(* CODESYS project øving 3.ecp

Project tree, tasks and I/O mapping:
  Controller : 750-8214 PFC200 G2 2ETH RS CAN, WAGO, order no. 0750-8214, version 5.16.3.16
    application Application
      libraries: 
      task PLC_Task (cyclic, interval t#50ms, priority 15) calls PLC_PRG, Oppgave4Teller, Oppgave3ST, Oppgave2BTest, Oppgave2ST
      task VISU_TASK (cyclic, interval 100 ms, priority 15) calls VisuElems.Visu_Prg
      program PLC_PRG [ST]
      global variables GVL
      Oppgave2/
        program Oppgave2ALD [LD]
        program Oppgave2ST [ST]
        program Oppgave2FBD [FBD]
        function Oppgave2A [FBD]
        function MFTest [FBD]
        function MLTest [LD]
        function MSTest [ST]
        function block RTF [FBD]
      Oppgave3/
        program Oppgave3LD [FBD]
        program Oppgave3FBD [FBD]
        program Oppgave3ST [FBD]
        function block Oppgave3STD [ST]
        function block Oppgave3FBDD [FBD]
        function block Oppgave3LDD [LD]
        visualisation Oppgave3GUI
      Oppgave4/
        function block Oppgave4Timeteller [ST]
        program Oppgave4Teller [FBD]
        visualisation Oppgave4Meny
      Oppgave2B/
        function Oppgave2B [ST]
        program Oppgave2BTest [ST]
      Oppgave1/
        program Oppgave1 [ST]
    ProjectConfigurationTxt
    ProjectConfiguration
    Kbus : Kbus, WAGO, version 1.4.0.2
        unmapped channels: K-BUS diagnostics
    MODBUS
      MODBUS : MODBUS, WAGO, order no. n/a, version 1.1.1.16
    CANbus
    Common.PCI
    EtherNet/IP
      Ethernet : Ethernet, WAGO, version 35.16.0.0
    Serial
      COM1 : COM1, WAGO, version 0.0.0.19
  00000000-0000-0000-0000-000000000000|C:\Users\kjebo\AppData\Local\Temp\4e63b915f46a404b8f25f3cc1ab48cd9\ProjectCfg.txt
  00000000-0000-0000-0000-000000000000|C:\Users\kjebo\AppData\Local\Temp\8f733436873c440eb71a6538c97844ea\Project.xml
  text list GlobalTextList
*)

// Controller/Application/GVL
{attribute 'qualified_only'}
VAR_GLOBAL
	Majority: BOOL;
	Vote1: BOOL;
	Vote2: BOOL;
	Vote3: BOOL;
	Trig: BOOL;
	Inn: BOOL;
	Ut: BOOL;
	
END_VAR

// Controller/Application/PLC_PRG
PROGRAM PLC_PRG
VAR
END_VAR

END_PROGRAM

// Controller/Application/Oppgave4/Oppgave4Teller
PROGRAM Oppgave4Teller
VAR
	Kjorer : BOOL;
	Time_ell: TIME;
	Timeteller_1: Oppgave4Timeteller;
	Omstart: BOOL;
	Alarm: BOOL; 
END_VAR

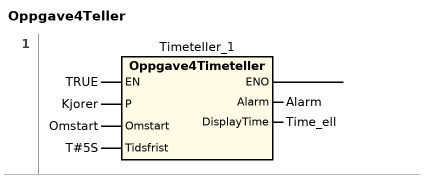
// NETWORK 1
Timeteller_1(P := Kjorer, Omstart := Omstart, Tidsfrist := T#5S, Alarm => Alarm, DisplayTime => Time_ell); // Oppgave4Timeteller

END_PROGRAM

// Controller/Application/Oppgave4/Oppgave4Timeteller
FUNCTION_BLOCK Oppgave4Timeteller
VAR_INPUT
	P: BOOL;
	Omstart: BOOL;
	Tidsfrist: TIME;
END_VAR
VAR_OUTPUT
	Alarm: BOOL;
	DisplayTime : TIME;
END_VAR
VAR
	T: TIME;
	T0: TIME;
	TT: TIME;
	StartTime: TIME;
	On: BOOL;
	P_A: BOOL;
	P_0: BOOL;
	Stopp: TIME;
	TotalRun : TIME;
	Sekunder: TIME;
END_VAR

P_A := P AND NOT (P_0);
P_0 := P;


//IF T0 = TIME() - TIME() THEN
	//T0 := TIME();
//END_IF
T := TIME();
IF On THEN
	//TT := TT + (T-T0);
	Sekunder := T - StartTime;
	IF T > Stopp THEN
		On := FALSE;
		TotalRun := Sekunder + TotalRun;
		Sekunder := T#0S;
		
	END_IF
ELSE 
	IF P_A THEN
		StartTime := T;
		TotalRun := Sekunder + TotalRun;
		Sekunder := T#0S;
		Stopp := StartTime + Tidsfrist;
		On := TRUE;
	END_IF
	
END_IF
T0 := T;
Displaytime := TotalRun + Sekunder;

IF T >= Stopp THEN
	Alarm := TRUE;
ELSE
	Alarm := FALSE;
END_IF

// Reset
IF Omstart THEN
	DisplayTime := T#0S;
	TotalRun := T#0s;
END_IF

END_FUNCTION_BLOCK

// Controller/Application/Oppgave3/Oppgave3ST
PROGRAM Oppgave3ST
VAR
	Oppgave3ST_0: Oppgave3STD;
END_VAR

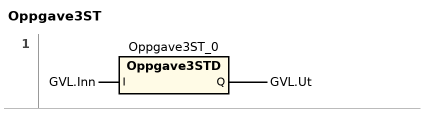
// NETWORK 1
Oppgave3ST_0(I := GVL.Inn); // Oppgave3STD
GVL.Ut := Oppgave3ST_0.Q;

END_PROGRAM

// Controller/Application/Oppgave3/Oppgave3STD
FUNCTION_BLOCK Oppgave3STD
VAR_INPUT
	I: BOOL;
END_VAR
VAR_OUTPUT
	Q: BOOL;
END_VAR
VAR
	PF: BOOL;
	I0: BOOL;
	Q0: BOOL;
END_VAR

PF := I AND NOT I0;
Q := PF XOR Q0;
Q0 := Q;
I0 := I;

END_FUNCTION_BLOCK

// Controller/Application/Oppgave2B/Oppgave2BTest
PROGRAM Oppgave2BTest
VAR
	Varme : REAL;
END_VAR

Varme := Oppgave2B(0 , 0 , 32767 , -20 , 300);

END_PROGRAM

// Controller/Application/Oppgave2B/Oppgave2B
FUNCTION Oppgave2B : REAL
VAR_INPUT
	Inn_Verdi : REAL;
	Inn_Min : REAL;
	Inn_Max : REAL;
	Ut_Min : REAL;
	Ut_Max : REAL;
END_VAR
VAR
	Valid : BOOL;
END_VAR

IF (Inn_Min<=Inn_Verdi AND Inn_Verdi<=Inn_Max AND Ut_Min<=Oppgave2B AND Oppgave2B<=Ut_Max)THEN
	Valid := TRUE;
	IF Valid = TRUE THEN
		Oppgave2B := (Inn_Verdi * ((Ut_Max - Ut_Min)/(Inn_Max - Inn_Min)))+Ut_Min;
	END_IF;
ELSE Oppgave2B := 0000000000000000000000000;
END_IF;

END_FUNCTION

// Controller/Application/Oppgave2/Oppgave2ST
PROGRAM Oppgave2ST
VAR
END_VAR

GVL.Majority := MSTest(GVL.Vote1, GVL.Vote2, GVL.Vote3);

END_PROGRAM

// Controller/Application/Oppgave2/MSTest
FUNCTION MSTest : BOOL
VAR_INPUT
	In1: BOOL;
	In2: BOOL;
	In3: BOOL;
END_VAR
VAR
END_VAR

IF (In1 = TRUE AND In2 = TRUE) OR (In1 = TRUE AND In3 = TRUE) OR (In2 = TRUE AND In3 = TRUE) THEN
	MSTest := TRUE;
ELSE
	MSTest := FALSE;
END_IF;

END_FUNCTION

// Controller/Application/Oppgave2/Oppgave2ALD
PROGRAM Oppgave2ALD
VAR
END_VAR

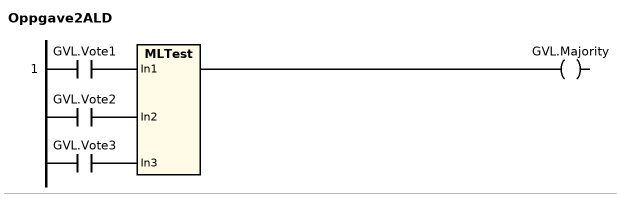
// NETWORK 1
GVL.Majority := MLTest(In1 := GVL.Vote1, In2 := GVL.Vote2, In3 := GVL.Vote3);

END_PROGRAM

// Controller/Application/Oppgave2/MLTest
FUNCTION MLTest : BOOL
VAR_INPUT
	In1 : BOOL;
	In2 : BOOL;
	In3 : BOOL;
END_VAR
VAR
END_VAR

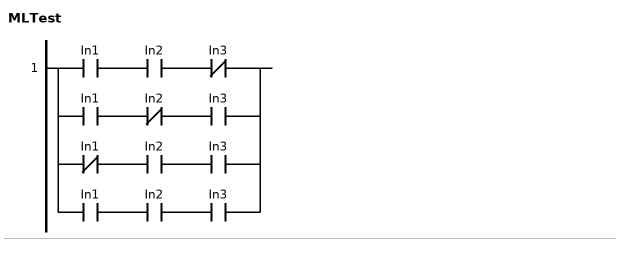
// NETWORK 1
(* In1 AND In2 AND NOT In3 OR In1 AND NOT In2 AND In3 OR NOT In1 AND In2 AND In3 OR In1 AND In2 AND In3; result not used *)

END_FUNCTION

// Controller/Application/Oppgave2/Oppgave2FBD
PROGRAM Oppgave2FBD
VAR
	Power: BOOL;
	Lamp: BOOL;
	RTF_0 : RTF;
END_VAR

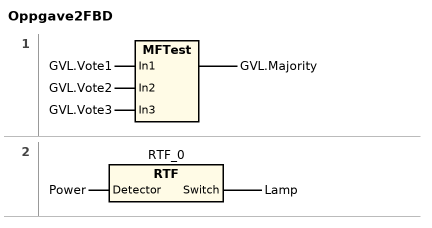
// NETWORK 1
GVL.Majority := MFTest(In1 := GVL.Vote1, In2 := GVL.Vote2, In3 := GVL.Vote3);

// NETWORK 2
RTF_0(Detector := Power); // RTF
Lamp := RTF_0.Switch;

END_PROGRAM

// Controller/Application/Oppgave2/MFTest
FUNCTION MFTest : BOOL
VAR_INPUT
	In1: BOOL;
	In2: BOOL;
	In3: BOOL;
END_VAR
VAR
END_VAR

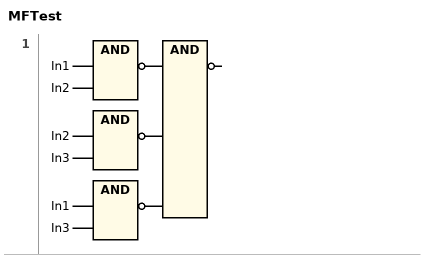
// NETWORK 1
(* NOT (In1 AND In2) AND NOT (In2 AND In3) AND NOT (In1 AND In3); result not used *)

END_FUNCTION

// Controller/Application/Oppgave2/RTF
FUNCTION_BLOCK RTF
VAR_INPUT
	Detector: BOOL;
END_VAR
VAR_OUTPUT
	Switch: BOOL;
END_VAR
VAR
	SR_0: SR;
	Trig1: R_TRIG;
	SR1: RS;
	Trig0: R_TRIG;
END_VAR

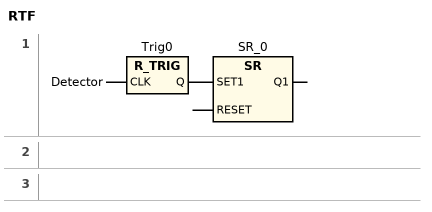
// NETWORK 1
Trig0(CLK := Detector); // R_TRIG
SR_0(SET1 := Trig0.Q); // SR

// NETWORK 2

// NETWORK 3

END_FUNCTION_BLOCK

// Controller/Application/Oppgave3/Oppgave3LD
PROGRAM Oppgave3LD
VAR
	Oppgave3LDD_0: Oppgave3LDD;
END_VAR

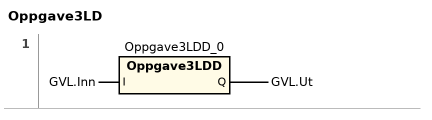
// NETWORK 1
Oppgave3LDD_0(I := GVL.Inn); // Oppgave3LDD
GVL.Ut := Oppgave3LDD_0.Q;

END_PROGRAM

// Controller/Application/Oppgave3/Oppgave3LDD
FUNCTION_BLOCK Oppgave3LDD
VAR_INPUT
	I: BOOL;
END_VAR
VAR_OUTPUT
	Q: BOOL;
END_VAR
VAR
	PF: BOOL;
	I0: BOOL;
	Q0: BOOL;
	SR_0: SR;
	SR_1: SR;
	SR_2: SR;
END_VAR

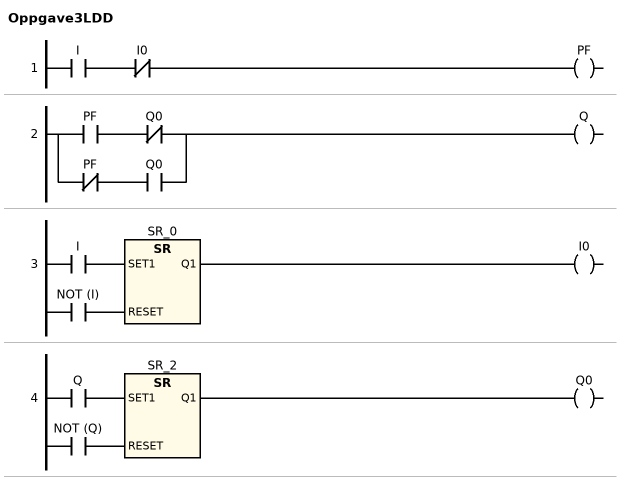
// NETWORK 1
PF := I AND NOT I0;

// NETWORK 2
Q := PF AND NOT Q0 OR NOT PF AND Q0;

// NETWORK 3
SR_0(SET1 := I, RESET := NOT (I)); // SR
I0 := SR_0.Q1;

// NETWORK 4
SR_2(SET1 := Q, RESET := NOT (Q)); // SR
Q0 := SR_2.Q1;

END_FUNCTION_BLOCK

// Controller/Application/Oppgave3/Oppgave3FBD
PROGRAM Oppgave3FBD
VAR
	Oppgave3FBD_0: Oppgave3FBDD;
END_VAR

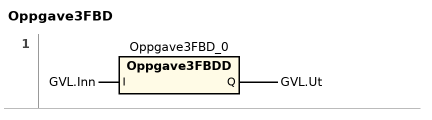
// NETWORK 1
Oppgave3FBD_0(I := GVL.Inn); // Oppgave3FBDD
GVL.Ut := Oppgave3FBD_0.Q;

END_PROGRAM

// Controller/Application/Oppgave3/Oppgave3FBDD
FUNCTION_BLOCK Oppgave3FBDD
VAR_INPUT
	I: BOOL;
END_VAR
VAR_OUTPUT
	Q: BOOL;
END_VAR
VAR
	I0: BOOL;
	
	Q0: BOOL;
	SR_I0: SR;
	SR_Q0: SR;
END_VAR

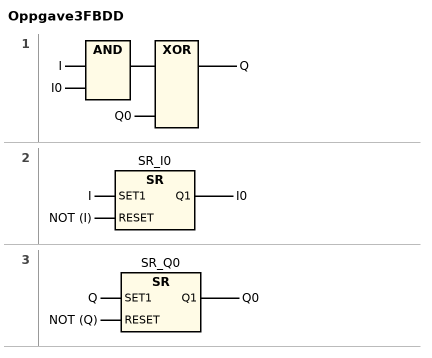
// NETWORK 1
Q := I AND I0 XOR Q0;

// NETWORK 2
SR_I0(SET1 := I, RESET := NOT (I)); // SR
I0 := SR_I0.Q1;

// NETWORK 3
SR_Q0(SET1 := Q, RESET := NOT (Q)); // SR
Q0 := SR_Q0.Q1;

END_FUNCTION_BLOCK

// Controller/Application/Oppgave1/Oppgave1
PROGRAM Oppgave1
VAR
END_VAR

//Forskjellen mellom funksjonsblokker og funksjoner er AT funksjonsblokker har minne mens funksjoner har ikke.
//Det vil si funksjoner gir samme resultat hver gang.
//Funksjonsblokker derimot husker hver gang den blir interacta med og kan derfor få forskjellige resultat
//mellom forskjellige bruk. 
//En POU er en funksjon\funksjonsblokk som kan opererer med flere verdier.

END_PROGRAM

// Controller/Application/Oppgave2/Oppgave2A
FUNCTION Oppgave2A : BOOL
VAR_INPUT
	Vote1 : BOOL;
	Vote2 : BOOL;
	Vote3 : BOOL;
END_VAR
VAR
END_VAR

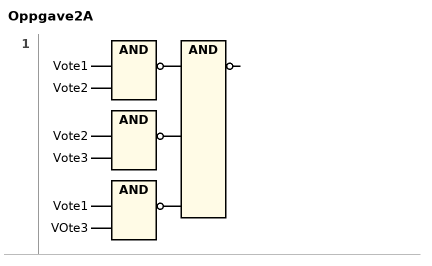
// NETWORK 1
(* NOT (Vote1 AND Vote2) AND NOT (Vote2 AND Vote3) AND NOT (Vote1 AND VOte3); result not used *)

END_FUNCTION

// Controller/Application/Oppgave3/Oppgave3GUI
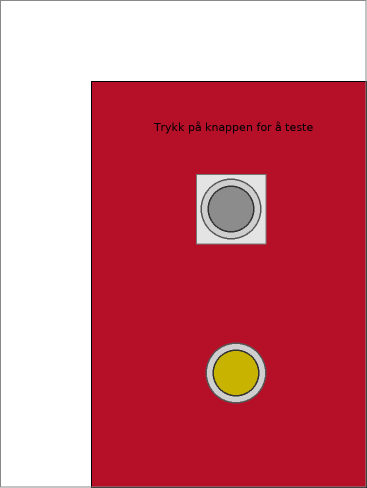
VISUALIZATION Oppgave3GUI  // 367x488
    Rectangle (91,81 276x407)
    Lamp1 (201,338 70x70), variable: GVL.Ut, style: Lamp-Lamp1-Yellow
    PushSwitch (196,174 70x70), variable: GVL.Inn, behaviour: TOGGLE, style: Switch-PushSwitch-Gray
    Label (134,101 200x53), "Trykk på knappen for å teste"
END_VISUALIZATION

// Controller/Application/Oppgave4/Oppgave4Meny
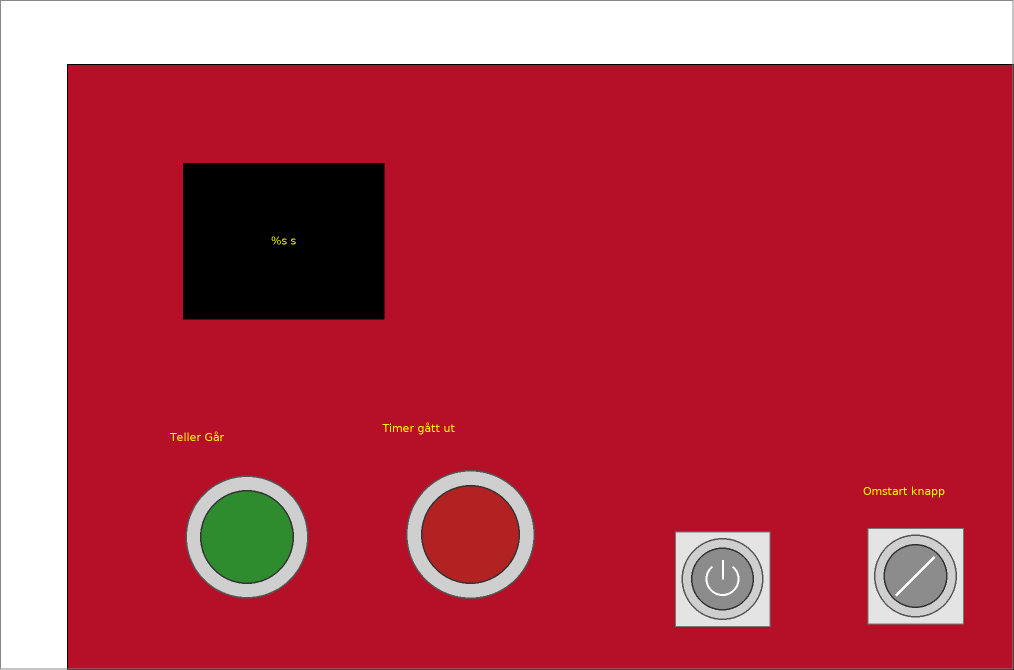
VISUALIZATION Oppgave4Meny  // 1014x670
    Rectangle (67,64 947x606)
    RotarySwitch (861,528 109x96), variable: Oppgave4Teller.Omstart, behaviour: TOGGLE, style: Switch-RotarySwitch-Gray
    Label (817,461 174x61), "Omstart knapp"
    Lamp1 (121,466 252x142), variable: Oppgave4Teller.Kjorer, style: Lamp-Lamp1-Green
    Lamp1 (352,460 237x149), variable: Oppgave4Teller.Alarm, style: Lamp-Lamp1-Red
    Label (336,406 169x45), "Timer gått ut"
    Label (111,411 172x53), "Teller Går"
    Rectangle (183,163 201x156), "%s s", text variable: Oppgave4Teller.Time_ell
    PowerSwitch (675,528 95x102), variable: Oppgave4Teller.Kjorer, behaviour: TOGGLE, style: Switch-PowerSwitch-Gray
END_VISUALIZATION
